{attribute 'linkalways'} 
{attribute 'no_explicit_call' := 'This FB is a CLASS and must be accessed using methods or properties'}
{attribute 'enable_dynamic_creation'}
FUNCTION_BLOCK _ETcVnDrawMatchesFlags EXTENDS EnumDatatypeBase
VAR
	localData : ETcVnDrawMatchesFlags;
	activeData : REFERENCE TO ETcVnDrawMatchesFlags;
	enumBaseDatatype : _DINT(localData);
END_VAR

METHOD PRIVATE AddLocalEnumeration
VAR_INPUT
	Enumeration : T_MAXSTRING;
	Value : ETcVnDrawMatchesFlags;
END_VAR
AddEnumeration(Enumeration, Value);
END_METHOD

PROPERTY PUBLIC Address : PVOID
GET
Address := ADR(activeData);
END_GET
END_PROPERTY

METHOD PUBLIC ClearReference
VAR_INPUT
END_VAR
activeData REF= localData;
SetBaseDatatypeReference();
END_METHOD

METHOD PUBLIC Clone : I_Datatype
VAR
    pClone : POINTER TO _ETcVnDrawMatchesFlags;
END_VAR
pClone := __NEW(_ETcVnDrawMatchesFlags(InitialValue := Value));
Clone := pClone^;
END_METHOD

METHOD FB_init : BOOL
VAR_INPUT
	bInitRetains : BOOL; // if TRUE, the retain variables are initialized (warm start / cold start)
	bInCopyCode : BOOL;  // if TRUE, the instance afterwards gets moved into the copy code (online change)
	InitialValue : ETcVnDrawMatchesFlags;
END_VAR
localData := InitialValue;
AddBaseDatatype(enumBaseDatatype);
ClearReference();

AddLocalEnumeration('TCVN_DMF_DEFAULT', ETcVnDrawMatchesFlags.TCVN_DMF_DEFAULT);
AddLocalEnumeration('TCVN_DMF_OVERDRAW', ETcVnDrawMatchesFlags.TCVN_DMF_OVERDRAW);
AddLocalEnumeration('TCVN_DMF_SKIPSINGLE', ETcVnDrawMatchesFlags.TCVN_DMF_SKIPSINGLE);
AddLocalEnumeration('TCVN_DMF_OVERDRAW_SKIPSINGLE', ETcVnDrawMatchesFlags.TCVN_DMF_OVERDRAW_SKIPSINGLE);
AddLocalEnumeration('TCVN_DMF_RICHKEYPOINT', ETcVnDrawMatchesFlags.TCVN_DMF_RICHKEYPOINT);
AddLocalEnumeration('TCVN_DMF_OVERDRAW_RICHKEYPOINT', ETcVnDrawMatchesFlags.TCVN_DMF_OVERDRAW_RICHKEYPOINT);
AddLocalEnumeration('TCVN_DMF_SKIPSINGLE_RICHKEYPOINT', ETcVnDrawMatchesFlags.TCVN_DMF_SKIPSINGLE_RICHKEYPOINT);
AddLocalEnumeration('TCVN_DMF_OVERDRAW_SKIPSINGLE_RICHKEYPOINT', ETcVnDrawMatchesFlags.TCVN_DMF_OVERDRAW_SKIPSINGLE_RICHKEYPOINT);
END_METHOD

PROPERTY PUBLIC Identifier : T_MAXSTRING
GET
Identifier := 'ETcVnDrawMatchesFlags';
END_GET
END_PROPERTY

METHOD IsEnumeratorValueEqual : BOOL
VAR_INPUT
	Enumerator : I_KeyValueForwardEnumerator;
END_VAR
VAR
	storedValue : ETcVnDrawMatchesFlags;
END_VAR
IF NOT Enumerator.TryGet(storedValue) THEN
	RETURN;
END_IF

IsEnumeratorValueEqual := storedValue = activeData;
END_METHOD

METHOD PUBLIC MakeReferenceTo
VAR_INPUT
	ReferenceTarget : REFERENCE TO ETcVnDrawMatchesFlags;
END_VAR
activeData REF= ReferenceTarget;
SetBaseDatatypeReference();
END_METHOD

METHOD PROTECTED SetBaseDatatypeReference
VAR_INPUT
END_VAR
enumBaseDatatype.MakeReferenceTo(activeData);
END_METHOD

PROPERTY PUBLIC Size : UDINT
GET
Size := SIZEOF(activeData);
END_GET
END_PROPERTY

METHOD TryMakeReferenceTo : BOOL
VAR_INPUT
	Target : I_Datatype;
END_VAR
VAR
	pTargetData : POINTER TO ETcVnDrawMatchesFlags;
END_VAR
IF NOT IsEquivalentTo(Target) THEN
	RETURN;
END_IF

pTargetData := Target.Address;
activeData REF= pTargetData^;
SetBaseDatatypeReference();
TryMakeReferenceTo := TRUE;
END_METHOD

PROPERTY PUBLIC Value : ETcVnDrawMatchesFlags
GET
Value := activeData;
END_GET
SET
activeData := Value;
END_SET
END_PROPERTY

END_FUNCTION_BLOCK

(* stored: Version 1.1.0.1, ProductVersion 3.1.4024.13
   POU _ETcVnDrawMatchesFlags: Id {e969a346-2e52-0295-2375-7b616dc979de}, SpecialFunc None
   Folder Core: Id {798faa80-0a02-076d-2ad0-a8c09c16d7ea}
   Folder Protected: Id {13738084-bad8-03dd-33af-d88fb66fa71e}
   Folder Customize: Id {7f148000-30c8-0442-15af-aa7dcd8b3869}
   Folder Constructor: Id {a8d25a69-e6ff-0d1f-27d5-1063947a0e79}
   Folder Private: Id {5c8b8169-756c-0dbc-18e8-9bcb70ff4eb4}
   Folder Protected: Id {7f0da98a-5d0c-0edd-0f17-4dfd99cb7b32}
   Method AddLocalEnumeration: Id {40c320ef-184e-01b7-1f2b-5bb5c6bd3058}
   Property Address: Id {9c1e89d3-8b07-0490-096b-444b7e2dc60b}
   Get Get: Id {b9976b3f-7c68-0394-33a4-433e7e0c6d56}
   Method ClearReference: Id {d78d9a97-1677-0013-0138-5eae598cab03}
   Method Clone: Id {7dc295ed-d27e-0a50-0da4-f6fea6bc9bc3}
   Method FB_init: Id {43aee692-4d4a-0dd0-1bea-a152b0d3f208}
   Property Identifier: Id {86487d81-73c7-0f49-1f99-92e183dbbc1b}
   Get Get: Id {ce1791fe-4545-0da1-3413-962fa4982027}
   Method IsEnumeratorValueEqual: Id {c0d7ea0c-e29d-0668-2137-c6496333e272}
   Method MakeReferenceTo: Id {7edf67e5-c864-09b1-27d7-044d99859a3a}
   Method SetBaseDatatypeReference: Id {34e767b0-e260-0181-07ec-5d07952655aa}
   Property Size: Id {7f7c2f64-c03d-0edf-14f1-2c6bfb5bde68}
   Get Get: Id {6c53df6c-b37b-0819-24cc-a81448ddb75d}
   Method TryMakeReferenceTo: Id {2027459d-4f84-03fe-1b84-35123d722093}
   Property Value: Id {92de1790-fafd-0a83-21e9-d603d5c10cf8}
   Get Get: Id {27b3463e-5e4d-04fd-10b9-848ef7dc1aaf}
   Set Set: Id {274df711-f41f-039c-00ab-aa909363275c} *)
